Fanuc KAREL source: kf00096.KL

-- PROVISIONAL review KL for V770-1; original PC SHA256 fb7610fc163bcbb5504bdf29b8da87790adc4ef101e31dbe342e150acca1a2ff
-- Incomplete behavior may be omitted. Consult companion uncertainty JSON. Do not deploy.
PROGRAM KF00096
%NOLOCKGROUP
BEGIN
  -- UNRESOLVED_PC offsets 5-16; opcodes 2E,23
  -- UNRESOLVED_PC offsets 21-32; opcodes 2E,23
  -- UNRESOLVED_PC offsets 37-67; opcodes 27,27,9D,22,22,22,22,31
  -- UNRESOLVED_PC offsets 72-76; opcodes 7F
END KF00096
